// Mitsubishi GX Works2 project: 2023-04-27 #2 생산자동화기능사 1번   PLC: Q03UDV

// global labels: Global1
VAR_GLOBAL
  PB1 AT X0 : BOOL;
  PB2 AT X1 : BOOL;
  정지 AT X2 : BOOL;
  공급후진 AT X3 : BOOL;
  공급전진 AT X4 : BOOL;
  가공후진 AT X5 : BOOL;
  가공전진 AT X6 : BOOL;
  송출후진 AT X7 : BOOL;
  송출전진 AT X8 : BOOL;
  배출후진 AT X9 : BOOL;
  배출전진 AT X0A : BOOL;
  매거진 AT X0B : BOOL;
  PB3 AT X0D : BOOL;
  금속센서 AT X0F : BOOL;
  적색 AT Y20 : BOOL;
  황색 AT Y21 : BOOL;
  녹색 AT Y22 : BOOL;
  공급1 AT Y23 : BOOL;
  공급2 AT Y24 : BOOL;
  가공 AT Y25 : BOOL;
  드릴 AT Y26 : BOOL;
  송출 AT Y27 : BOOL;
  배출 AT Y28 : BOOL;
  컨베이어 AT Y29 : BOOL;
END_VAR

PROGRAM 테스트동작
VAR
  STATE : INT;
END_VAR
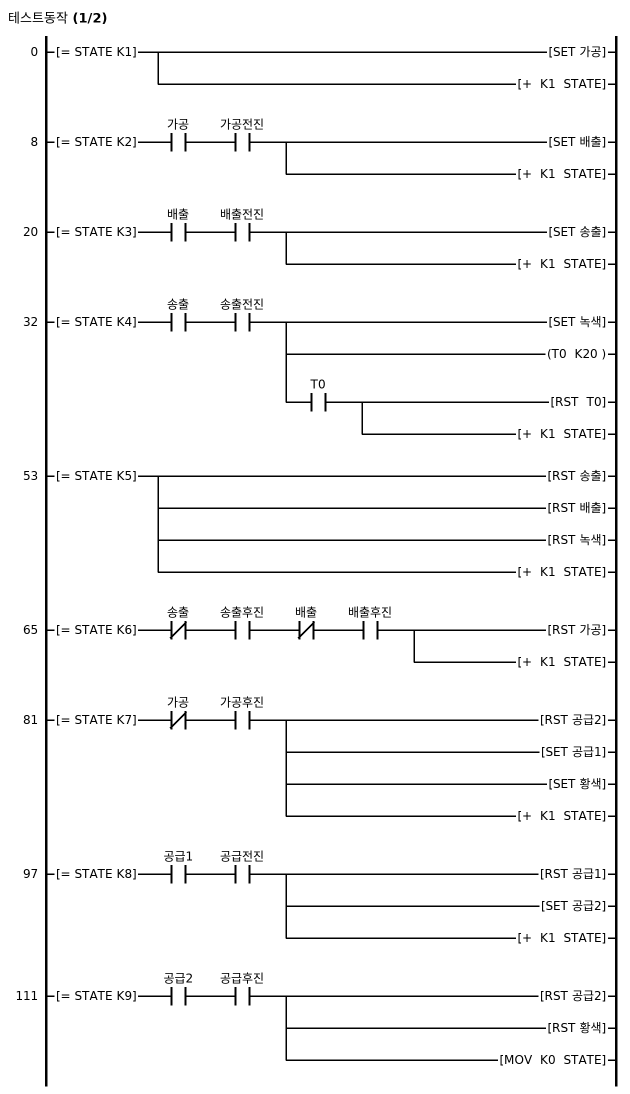
0     LD=     STATE K1
      SET     가공
      +       K1 STATE
8     LD=     STATE K2
      AND     가공
      AND     가공전진
      SET     배출
      +       K1 STATE
20    LD=     STATE K3
      AND     배출
      AND     배출전진
      SET     송출
      +       K1 STATE
32    LD=     STATE K4
      AND     송출
      AND     송출전진
      SET     녹색
      OUT     T0 K20
      AND     T0
      RST     T0
      +       K1 STATE
53    LD=     STATE K5
      RST     송출
      RST     배출
      RST     녹색
      +       K1 STATE
65    LD=     STATE K6
      ANI     송출
      AND     송출후진
      ANI     배출
      AND     배출후진
      RST     가공
      +       K1 STATE
81    LD=     STATE K7
      ANI     가공
      AND     가공후진
      RST     공급2
      SET     공급1
      SET     황색
      +       K1 STATE
97    LD=     STATE K8
      AND     공급1
      AND     공급전진
      RST     공급1
      SET     공급2
      +       K1 STATE
111   LD=     STATE K9
      AND     공급2
      AND     공급후진
      RST     공급2
      RST     황색
      MOV     K0 STATE
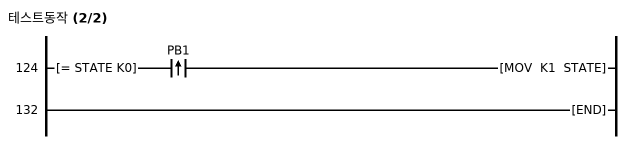
124   LD=     STATE K0
      ANDP    PB1
      MOV     K1 STATE
132   END
END_PROGRAM

PROGRAM 단속동작
VAR
  STATE : INT;
END_VAR
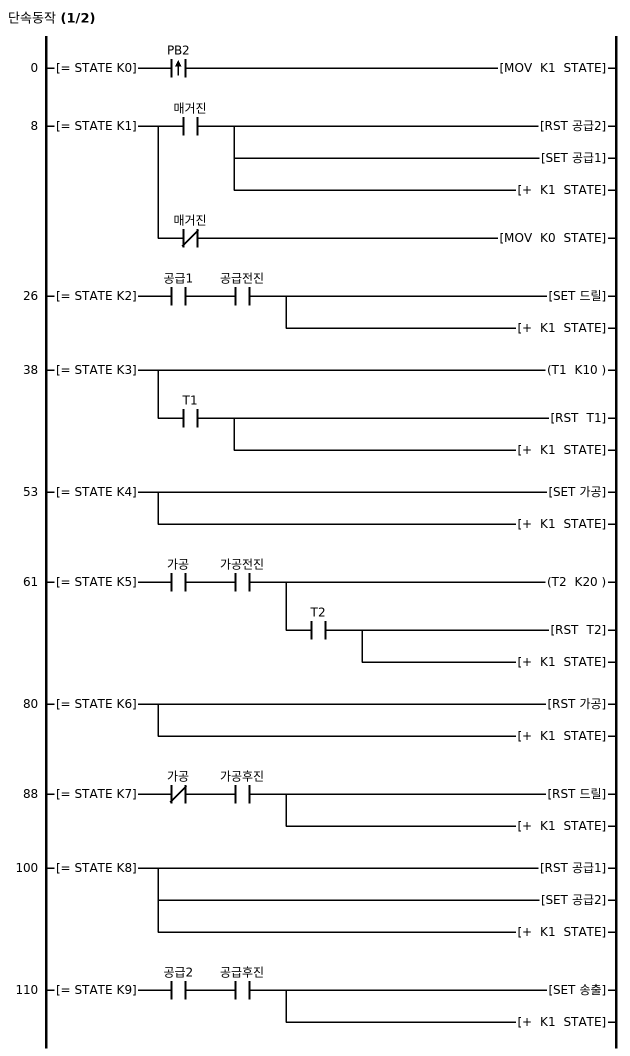
0     LD=     STATE K0
      ANDP    PB2
      MOV     K1 STATE
8     LD=     STATE K1
      MPS
      AND     매거진
      RST     공급2
      SET     공급1
      +       K1 STATE
      MPP
      ANI     매거진
      MOV     K0 STATE
26    LD=     STATE K2
      AND     공급1
      AND     공급전진
      SET     드릴
      +       K1 STATE
38    LD=     STATE K3
      OUT     T1 K10
      AND     T1
      RST     T1
      +       K1 STATE
53    LD=     STATE K4
      SET     가공
      +       K1 STATE
61    LD=     STATE K5
      AND     가공
      AND     가공전진
      OUT     T2 K20
      AND     T2
      RST     T2
      +       K1 STATE
80    LD=     STATE K6
      RST     가공
      +       K1 STATE
88    LD=     STATE K7
      ANI     가공
      AND     가공후진
      RST     드릴
      +       K1 STATE
100   LD=     STATE K8
      RST     공급1
      SET     공급2
      +       K1 STATE
110   LD=     STATE K9
      AND     공급2
      AND     공급후진
      SET     송출
      +       K1 STATE
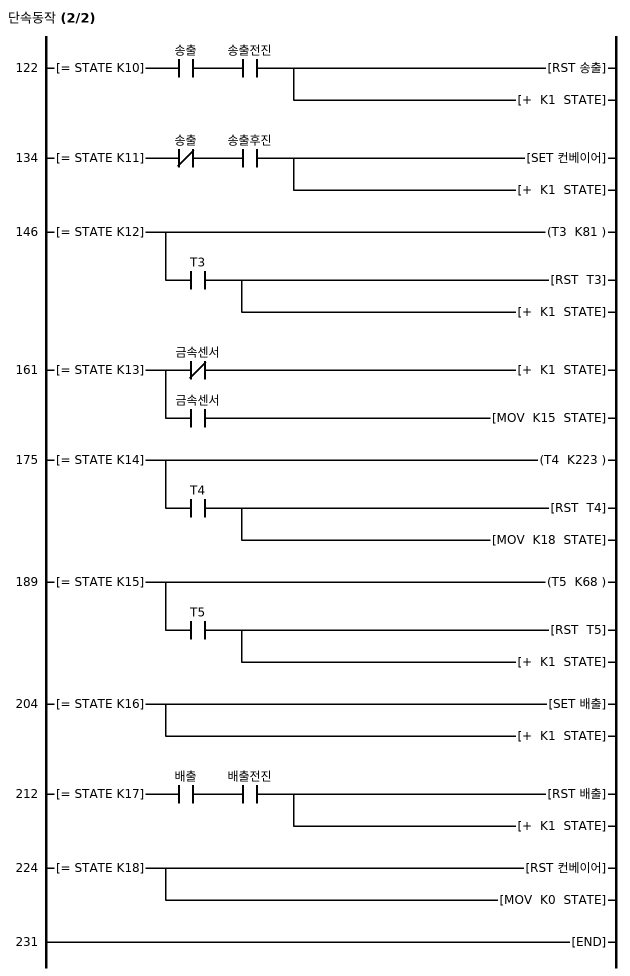
122   LD=     STATE K10
      AND     송출
      AND     송출전진
      RST     송출
      +       K1 STATE
134   LD=     STATE K11
      ANI     송출
      AND     송출후진
      SET     컨베이어
      +       K1 STATE
146   LD=     STATE K12
      OUT     T3 K81
      AND     T3
      RST     T3
      +       K1 STATE
161   LD=     STATE K13
      MPS
      ANI     금속센서
      +       K1 STATE
      MPP
      AND     금속센서
      MOV     K15 STATE
175   LD=     STATE K14
      OUT     T4 K223
      AND     T4
      RST     T4
      MOV     K18 STATE
189   LD=     STATE K15
      OUT     T5 K68
      AND     T5
      RST     T5
      +       K1 STATE
204   LD=     STATE K16
      SET     배출
      +       K1 STATE
212   LD=     STATE K17
      AND     배출
      AND     배출전진
      RST     배출
      +       K1 STATE
224   LD=     STATE K18
      RST     컨베이어
      MOV     K0 STATE
231   END
END_PROGRAM

PROGRAM 연속동작
VAR
  STATE : INT;
END_VAR
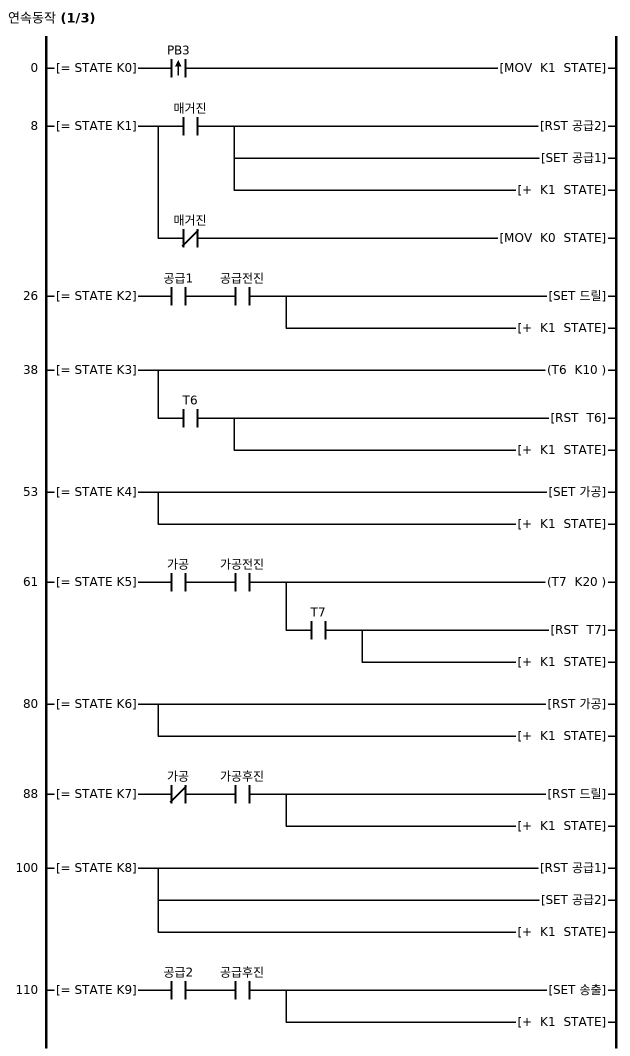
0     LD=     STATE K0
      ANDP    PB3
      MOV     K1 STATE
8     LD=     STATE K1
      MPS
      AND     매거진
      RST     공급2
      SET     공급1
      +       K1 STATE
      MPP
      ANI     매거진
      MOV     K0 STATE
26    LD=     STATE K2
      AND     공급1
      AND     공급전진
      SET     드릴
      +       K1 STATE
38    LD=     STATE K3
      OUT     T6 K10
      AND     T6
      RST     T6
      +       K1 STATE
53    LD=     STATE K4
      SET     가공
      +       K1 STATE
61    LD=     STATE K5
      AND     가공
      AND     가공전진
      OUT     T7 K20
      AND     T7
      RST     T7
      +       K1 STATE
80    LD=     STATE K6
      RST     가공
      +       K1 STATE
88    LD=     STATE K7
      ANI     가공
      AND     가공후진
      RST     드릴
      +       K1 STATE
100   LD=     STATE K8
      RST     공급1
      SET     공급2
      +       K1 STATE
110   LD=     STATE K9
      AND     공급2
      AND     공급후진
      SET     송출
      +       K1 STATE
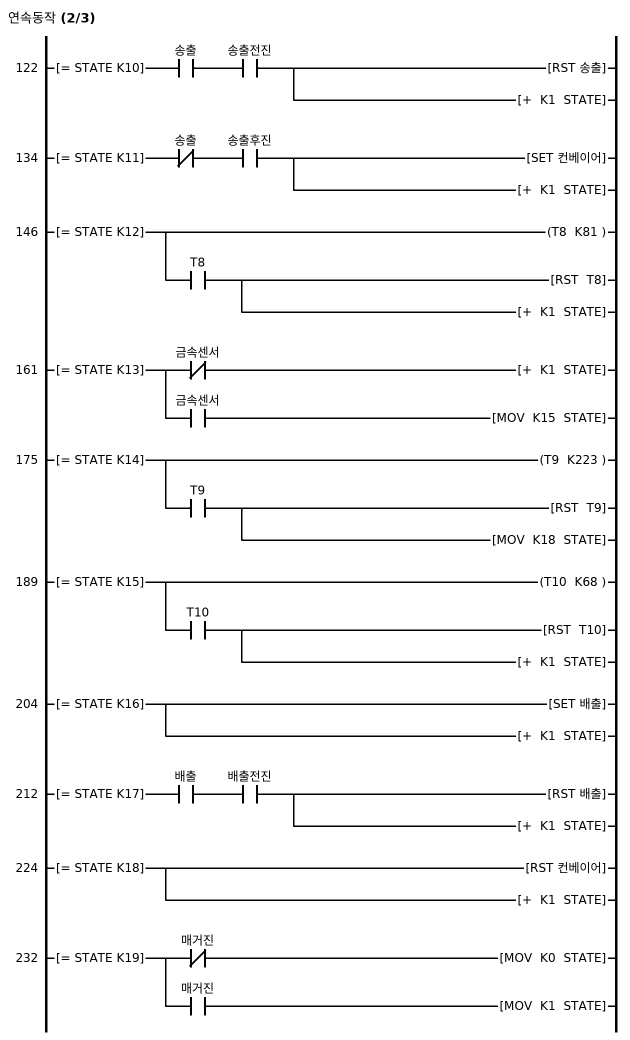
122   LD=     STATE K10
      AND     송출
      AND     송출전진
      RST     송출
      +       K1 STATE
134   LD=     STATE K11
      ANI     송출
      AND     송출후진
      SET     컨베이어
      +       K1 STATE
146   LD=     STATE K12
      OUT     T8 K81
      AND     T8
      RST     T8
      +       K1 STATE
161   LD=     STATE K13
      MPS
      ANI     금속센서
      +       K1 STATE
      MPP
      AND     금속센서
      MOV     K15 STATE
175   LD=     STATE K14
      OUT     T9 K223
      AND     T9
      RST     T9
      MOV     K18 STATE
189   LD=     STATE K15
      OUT     T10 K68
      AND     T10
      RST     T10
      +       K1 STATE
204   LD=     STATE K16
      SET     배출
      +       K1 STATE
212   LD=     STATE K17
      AND     배출
      AND     배출전진
      RST     배출
      +       K1 STATE
224   LD=     STATE K18
      RST     컨베이어
      +       K1 STATE
232   LD=     STATE K19
      MPS
      ANI     매거진
      MOV     K0 STATE
      MPP
      AND     매거진
      MOV     K1 STATE
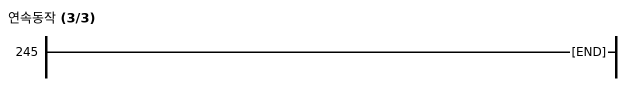
245   END
END_PROGRAM

PROGRAM 부가조건1
0     END
END_PROGRAM
